FUNCTION_BLOCK RT_Bridge_6 (* Data connection decoupling bridge for data connection between real-time event chains *)
  (* Standard: 61499-2; Description: Copyright (c) 2023 Johannes Kepler University Linz This program and the accompanying materials are made available under the terms of the Eclipse Public License 2.0 which is available at https://www.eclipse.org/legal/epl-2.0/ SPDX-License-Identifier: EPL-2.0 *)
  (* Version 3.0, 2025-04-14, Patrick Aigner, changed package *)
  (* Version 1.0, 2023-11-02, Alois Zoitl, Johannes Kepler University Linz *)
  PACKAGE eclipse4diac::rtevents;
  {SET_ATTRIBUTE(eclipse4diac::core::GenericClassName, 'GEN_RT_Bridge')}
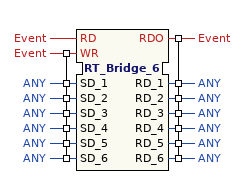
  EVENT_INPUT
    RD; (* Read data from data bridge *)
    WR WITH SD_1, SD_2, SD_3, SD_4, SD_5, SD_6; (* Write data to data bridge *)
  END_EVENT
  EVENT_OUTPUT
    RDO WITH RD_1, RD_2, RD_3, RD_4, RD_5, RD_6; (* Read data notifcation *)
  END_EVENT
  VAR_INPUT
    SD_1 : ANY; (* Data to be put into the data bridge *)
    SD_2 : ANY; (* Data to be put into the data bridge *)
    SD_3 : ANY; (* Data to be put into the data bridge *)
    SD_4 : ANY; (* Data to be put into the data bridge *)
    SD_5 : ANY; (* Data to be put into the data bridge *)
    SD_6 : ANY; (* Data to be put into the data bridge *)
  END_VAR
  VAR_OUTPUT
    RD_1 : ANY; (* Data from data bridge *)
    RD_2 : ANY; (* Data from data bridge *)
    RD_3 : ANY; (* Data from data bridge *)
    RD_4 : ANY; (* Data from data bridge *)
    RD_5 : ANY; (* Data from data bridge *)
    RD_6 : ANY; (* Data from data bridge *)
  END_VAR
END_FUNCTION_BLOCK
